# EPICS StreamDevice protocol: siteLibs/TC353LibSrc/proto/TC353.proto
# TC-353 Stream protocol file

Terminator = CR;
ReplyTimeout = 10000;
ReadTimeout = 1000;

crc_to_null {
    out "SCC0b98a!";
    in "$!";
}

start_bo {
    out "SDR%d!";
    in "$!";
}

oper_time_ai {
    out "RDT!";
    in "%d!";
}

read_status_mbbi {
    out "RSS!";
    in "%d!";
}

read_failure_ai {
    out "RSA!";
    in "#%d!";
    @mismatch {
        in "%d!";
    }
}

read_freq_ai {
    out "RRS!";
    in "%d!";
}
